PROGRAM ConnectSystem
VAR
	ConnectR1		:FB_Connection;
END_VAR

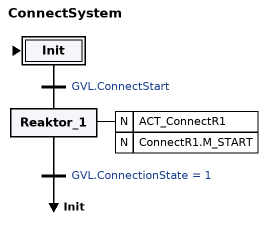
INITIAL_STEP Init:
END_STEP
TRANSITION FROM Init TO Reaktor_1
    := GVL.ConnectStart;
END_TRANSITION
STEP Reaktor_1:
    ACT_ConnectR1(N);
    ConnectR1.M_START(N);
END_STEP
TRANSITION FROM Reaktor_1 TO Init
    := GVL.ConnectionState = 1;
END_TRANSITION

ACTION ACT_ConnectR1:
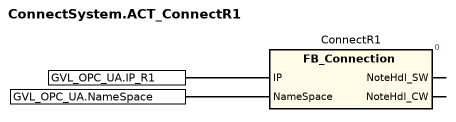
ConnectR1(IP := GVL_OPC_UA.IP_R1, NameSpace := GVL_OPC_UA.NameSpace); // FB_Connection
END_ACTION

END_PROGRAM

(* stored: Version 1.1.0.1, ProductVersion 3.1.4024.12
   POU ConnectSystem: Id {49677b0c-65b7-4c24-b2cc-6fac1dce0356}, SpecialFunc None
   Folder 01_Aktionen: Id {131982a0-b797-484f-8dad-6aea63ef6a17}
   Action ACT_ConnectR1: Id {31c538ec-1287-4a5a-b974-a1fd7db5c0ee} *)
